{attribute addProperty BoxType "EL3403-0000-0022"}
{attribute addProperty Id "PM_Inputs_ChannelAT %I*ARRAY[0..2] OF PM_Inputs_Channel_D07DCD53432540PM_Status_dataAT %I*PM_Status_data_F5918FB93240PM_Outputs_ChannelAT %Q*ARRAY[0..2] OF PM_Outputs_Channel_A1108FBB2430WcStateAT %I*WcState_F855686C1620InfoDataAT %I*InfoData_BC63D37F80100"}
{attribute addProperty CRC "1355284726"}
{attribute addProperty SizeInBites "584"}
{attribute addProperty SizeInBytes "73"}
TYPE EL3403_26274D99 :
STRUCT
	{attribute addProperty Name "PM_Inputs_Channel"}
	PM_Inputs_Channel : ARRAY[0..2] OF PM_Inputs_Channel_D07DCD53;
	{attribute addProperty Name "PM_Status_data"}
	PM_Status_data : PM_Status_data_F5918FB9;
	{attribute addProperty Name "PM_Outputs_Channel"}
	PM_Outputs_Channel : ARRAY[0..2] OF PM_Outputs_Channel_A1108FBB;
	{attribute addProperty Name "WcState"}
	WcState : WcState_F855686C;
	{attribute addProperty Name "InfoData"}
	InfoData : InfoData_BC63D37F;
END_STRUCT
END_TYPE

(* stored: Version 1.2.0.0, ProductVersion 3.1.4024.9
   DUT EL3403_26274D99: Id {f605ccd5-aca7-4259-977c-f74c1235bbb7} *)
